// TwinCAT 3 PLC project AdsStaticNetId
// ProgramVersion: 3.1.4023.0
// libraries:
//   Tc2_DataExchange, * (Beckhoff Automation GmbH)
//   Tc2_Standard, * (Beckhoff Automation GmbH)
//   Tc2_System, * (Beckhoff Automation GmbH)
//   Tc2_Utilities, * (Beckhoff Automation GmbH)
//   Tc3_BA_Common, * (Beckhoff Automation GmbH)
//   Tc3_Module, * (Beckhoff Automation GmbH)
// project tree:
//   DUTs/ AdsData.TcDUT (not stored), AdsMessageQueue.TcPOU, AdsMessage.TcDUT (not stored), AdsSocket.TcPOU, AreaNum.TcDUT (not stored), EventsEnum.TcTLEO (not stored)
//   GVLs/ LocalSocket.TcGVL (not stored)
//   / PlcTask.TcTTO (not stored)
//   POUs/ AdsTcp_WinStd.TcPOU, BufferIsEmpty.TcPOU, MAIN.TcPOU
// real-time tasks:
//   TASK PlcTask: cycle T#10ms, priority 21, ADS port 350

// ---- DUTs/AdsMessageQueue.TcPOU
{attribute 'call_after_init'}
FUNCTION_BLOCK AdsMessageQueue
VAR
	elements : FB_BA_DynamicArray := (uiEntrySize := SIZEOF(POINTER TO AdsMessage), uiMinExpCount := 4); 
	length : INT := 0;
	
	entrySize : UDINT;
END_VAR
(*
this container stores dynamically generated AdsData Structs
AdsData to be added are passed by reference, then this function block allocates a structure to be stored
AdsData are get() by reference and poll() by value
*)

METHOD clear : BOOL
VAR
	i : INT;
	temp : REFERENCE TO AdsMessage;
	tempAdr : POINTER TO AdsMessage;
END_VAR
FOR i:=0 TO length-1 BY 1 DO
	temp := get(index := i, getSize => );
	tempAdr := ADR(temp);
	__DELETE(tempAdr);
END_FOR

elements.Reset();
length := 0;
END_METHOD

METHOD contains : BOOL //check contents, not pointer value
VAR_INPUT
	value : REFERENCE TO AdsMessage;
END_VAR
VAR_OUTPUT
	atIndex : INT;
END_VAR
VAR
	temp : REFERENCE TO AdsMessage;
	i : INT;
END_VAR
IF length = 0 THEN
	contains := FALSE;
	RETURN;
END_IF

FOR i:=0 TO length-1 BY 1 DO
	temp := get(index := i, getSize => );
	
	IF 
		SIZEOF(value) = entrySize AND //same size
		MEMCMP(ADR(temp), ADR(value), SIZEOF(entrySize)) = 0 //same data
	THEN
		contains := TRUE;
		atIndex := i;
		RETURN;
	END_IF
	
END_FOR
contains := FALSE;
END_METHOD

METHOD get : REFERENCE TO AdsMessage
VAR_INPUT
	index : INT;
END_VAR
VAR_OUTPUT
	getSize : UDINT;
END_VAR
IF length = 0 OR index < 0 OR index >= length THEN
	getSize := 0;
ELSE
	elements.GetEntry(diIndex := index, pResultEntry := ADR(get));
	getSize := SIZEOF(get);
END_IF
END_METHOD

METHOD isEmpty : BOOL
VAR_INPUT
END_VAR
isEmpty := length = 0;
END_METHOD

METHOD poll : AdsMessage
VAR_OUTPUT
	getSize : UDINT;
END_VAR
IF length > 0 THEN
	poll := get(index := 0, getSize => getSize);
	elements.RemoveEntry(diIndex := 0);
	
	length := length - 1;
END_IF
END_METHOD

METHOD push : BOOL
VAR_INPUT
	value : REFERENCE TO AdsMessage;
END_VAR
VAR
	temp : POINTER TO AdsMessage;
END_VAR
temp := __NEW(AdsMessage);
temp^ := value;

elements.AddEntryPtr(pEntry := temp);

length := length + 1;
END_METHOD

METHOD set : BOOL
VAR_INPUT
	i : INT;
	value : REFERENCE TO AdsMessage;
END_VAR
VAR
	temp : REFERENCE TO AdsMessage;
END_VAR
IF length = 0 THEN
	RETURN;
END_IF

IF i >= 0 AND i < length THEN
	temp REF= get(i);
	temp := value;
	
	set := TRUE;
END_IF
END_METHOD

{attribute 'call_after_init'}
METHOD setup : BOOL
VAR_INPUT
END_VAR
entrySize := SIZEOF(AdsMessage);
END_METHOD

METHOD size : INT
size := length;
END_METHOD

END_FUNCTION_BLOCK

// ---- DUTs/AdsSocket.TcPOU
FUNCTION_BLOCK AdsSocket
VAR_INPUT
END_VAR
VAR_OUTPUT
	//descriptive string for the name of the running program, may or may not be used
	PrgName : STRING;
	
	(*
	AmsNetId should be in the following format for ALL Beckhoff PLCs in the network:
		<area number> . <subarea number (0 for master PLC)> .131.216.1.1
		panel PCs to be assigned 113.174 instead of 131.216
			2.0.131.216.1.1 - Area 2, master controller
			4.3.113.174.1.1 - Area 4, manual station 3 panel PC
	*)
	AmsNetId : T_AmsNetId;
	
	//for now, use ADS port 851 for communication
	AmsPort : T_AmsPort;
END_VAR
VAR_OUTPUT
	receivingData : AdsData;
	sendingData : AdsData;
	
	readBusy : BOOL;
	readError : BOOL;
	readErrorId : UDINT;
	
	writeBusy : BOOL;
	writeError : BOOL;
	writeErrorId : UDINT;
END_VAR
VAR	
	adsWriteSymbol : FB_WriteAdsSymByName;
	adsReadSymbol : FB_ReadAdsSymByName;
END_VAR
VAR
	targetSocket : STRING;
	clearing : BOOL;
END_VAR
(*
TCP-style ADS connection that only writes to a buffer in the recipient's AdsTcpUnit module
*)

//write into the recipient's allocated socket for this system
(*
IF FIND(AmsNetId, '113.174') > 0 THEN //panel PC
	targetSocket := CONCAT('AdsTcp_WinCE.', LocalSocket.PrgName);
ELSE//CX5130+ IPC
	targetSocket := CONCAT('AdsTcp_WinStd.', LocalSocket.PrgName);
END_IF
*)
targetSocket := CONCAT('AdsTcp_WinCE.', LocalSocket.PrgName);
//only toggles if data has contents, otherwise remains false
adsWriteSymbol.bWrite := NOT BufferIsEmpty(sendingData.binaryData) AND NOT adsWriteSymbol.bWrite;
(*
IF NOT BufferIsEmpty(sendingData.binaryData) THEN
	adsWriteSymbol.bWrite := NOT adsWriteSymbol.bWrite;
ELSE
	adsWriteSymbol.bWrite := FALSE;
END_IF 
*)
blocks();

IF NOT adsWriteSymbol.bBusy THEN
	MEMSET(ADR(sendingData), 0, SIZEOF(sendingData));
END_IF

METHOD PRIVATE blocks : BOOL
VAR_INPUT
END_VAR
adsReadSymbol(
	bRead:= , 
	sNetId:= AmsNetId, 
	nPort:= AmsPort, 
	sVarName:= , 
	nDestAddr:= , 
	nLen:= , 
	tTimeout:= , 
	eComMode:= , 
	bClearOnError:= , 
	bBusy=> readBusy, 
	bError=> readError, 
	nErrorId=> readErrorId);
	
adsWriteSymbol(
	bWrite:= , 
	sNetId:= AmsNetId, 
	nPort:= AmsPort, 
	sVarName:= CONCAT(targetSocket, '.receivingData'), 
	nSrcAddr:= ADR(sendingData), 
	nLen:= SIZEOF(sendingData), 
	tTimeout:= , 
	eComMode:= eAdsComModeSecureCom, 
	bBusy=> writeBusy, 
	bError=> writeError, 
	nErrorId=> writeErrorId);
END_METHOD

METHOD send : BOOL
VAR_INPUT
	data : REFERENCE TO AdsData;
END_VAR
sendingData := data;
END_METHOD

END_FUNCTION_BLOCK

// ---- POUs/BufferIsEmpty.TcPOU
FUNCTION BufferIsEmpty : BOOL
VAR_IN_OUT
	bufferArr : ARRAY[*] OF BYTE;
END_VAR
VAR
	i : DINT;
END_VAR

FOR i:=LOWER_BOUND(bufferArr, 1) TO UPPER_BOUND(bufferArr, 1) BY 1 DO
	IF bufferArr[i] <> 0 THEN
		BufferIsEmpty := FALSE;
		RETURN;
	END_IF
END_FOR
BufferIsEmpty := TRUE;

END_FUNCTION

// ---- POUs/AdsTcp_WinStd.TcPOU
PROGRAM AdsTcp_WinStd
VAR_OUTPUT
	bBusy : BOOL;
	err : BOOL;
	errid : UDINT;
END_VAR
VAR_OUTPUT
	areaSockets : ARRAY[1..6] OF POINTER TO AdsSocket; //only used for finding a socket by name, POINTER because array of REFERENCE does not exist
	
	//unlikely that each area will need communication with all other areas
	//only area 3 needs access to all areas, other areas only need access to area 3
	AREA_1 : AdsSocket := (PrgName := 'AREA_1', AmsNetId := '1.0.131.216.1.1', AmsPort := 851);
	AREA_2 : AdsSocket := (PrgName := 'AREA_2', AmsNetId := '2.0.131.216.1.1', AmsPort := 851);
	AREA_3 : AdsSocket := (PrgName := 'AREA_3', AmsNetId := '3.0.131.216.1.1', AmsPort := 851);
	AREA_4 : AdsSocket := (PrgName := 'AREA_4', AmsNetId := '4.0.131.216.1.1', AmsPort := 851);
	AREA_5 : AdsSocket := (PrgName := 'AREA_5', AmsNetId := '5.0.131.216.1.1', AmsPort := 851);
	AREA_6 : AdsSocket := (PrgName := 'AREA_6', AmsNetId := '6.0.131.216.1.1', AmsPort := 851);
END_VAR
VAR	
	tempSocket : REFERENCE TO AdsSocket;
	(*
	transmissons are queued into AdsTcpUnit, where all the preset sockets are
	to send a transmission, place the data and a recipient name into an AdsMessage type
	when a transmission is polled from the queue:
		if the recipient does not exist, the message contents are discarded
		if the recipient exists and is not busy writing, then the message contents are given to the socket to be written
		if the recipient is busy, then the messsage is pushed back into the queue
	*)
	transmissionQueue : AdsMessageQueue;
	nextTransmission : AdsMessage;
	
	i : INT(1..numSockets);
END_VAR
VAR CONSTANT
	numSockets : INT := 6-1;
END_VAR
(*
similar functionality to standard TCP communication - only writes to a single receiving buffer on the target system
	no read/write functionality to any other symbol on target
messages are entered into a queue which is polled cyclically and passed to the appropriate socket
*)

areaSockets[1] := ADR(AREA_1);
areaSockets[2] := ADR(AREA_2);
areaSockets[3] := ADR(AREA_3);
areaSockets[4] := ADR(AREA_4);
areaSockets[5] := ADR(AREA_5);
areaSockets[6] := ADR(AREA_6);

blocks();

nextTransmission := transmissionQueue.poll(getSize => );

tempSocket REF= findSocket(recipient := nextTransmission.recipient);

IF __ISVALIDREF(tempSocket) THEN
	
	IF NOT tempSocket.writeBusy THEN
		tempSocket.send(data := nextTransmission.contents);
	ELSE //if socket is busy, then message is returned to the end of the line
		transmissionQueue.push(value := nextTransmission);
	END_IF
	
END_IF
//if recipient does not exist, message is discarded

METHOD PRIVATE blocks : BOOL
VAR_INPUT
END_VAR
AREA_1(
	PrgName=> , 
	AmsNetId=> , 
	AmsPort=> , 
	receivingData=> , 
	sendingData=> , 
	readBusy=> , 
	readError=> , 
	readErrorId=> , 
	writeBusy=> , 
	writeError=> , 
	writeErrorId=> );

AREA_2(
	PrgName=> , 
	AmsNetId=> , 
	AmsPort=> , 
	receivingData=> , 
	sendingData=> , 
	readBusy=> , 
	readError=> , 
	readErrorId=> , 
	writeBusy=> , 
	writeError=> , 
	writeErrorId=> );
	
AREA_3(
	PrgName=> , 
	AmsNetId=> , 
	AmsPort=> , 
	receivingData=> , 
	sendingData=> , 
	readBusy=> , 
	readError=> , 
	readErrorId=> , 
	writeBusy=> , 
	writeError=> , 
	writeErrorId=> );
	
AREA_4(
	PrgName=> , 
	AmsNetId=> , 
	AmsPort=> , 
	receivingData=> , 
	sendingData=> , 
	readBusy=> , 
	readError=> , 
	readErrorId=> , 
	writeBusy=> , 
	writeError=> , 
	writeErrorId=> );
	
AREA_5(
	PrgName=> , 
	AmsNetId=> , 
	AmsPort=> , 
	receivingData=> , 
	sendingData=> , 
	readBusy=> , 
	readError=> , 
	readErrorId=> , 
	writeBusy=> , 
	writeError=> , 
	writeErrorId=> );
	
AREA_6(
	PrgName=> , 
	AmsNetId=> , 
	AmsPort=> , 
	receivingData=> , 
	sendingData=> , 
	readBusy=> , 
	readError=> , 
	readErrorId=> , 
	writeBusy=> , 
	writeError=> , 
	writeErrorId=> );
END_METHOD

METHOD PRIVATE findSocket : REFERENCE TO AdsSocket
VAR_INPUT
	recipient : STRING;
END_VAR
FOR i:=1 TO numSockets BY 1 DO
	IF areaSockets[i]^.PrgName = recipient THEN
		findSocket REF= areaSockets[i]^;
		RETURN;
	END_IF
END_FOR
END_METHOD

METHOD generateMessage : BOOL
VAR_INPUT
	recipient : STRING;
	description : EventsEnum;
	timestamp : TIMESTRUCT;
END_VAR
VAR_IN_OUT
	binaryData : ARRAY[*] OF BYTE;
END_VAR
VAR
	newTransmission : AdsMessage;
END_VAR
newTransmission.recipient := recipient;

newTransmission.contents.description := description;
newTransmission.contents.timestamp := timestamp;
MEMCPY(
	ADR(newTransmission.contents.binaryData),
	binaryData,
	MIN( TO_UDINT(UPPER_BOUND(binaryData, 1) - LOWER_BOUND(binaryData, 1) + 1), SIZEOF(newTransmission.contents.binaryData) ));
END_METHOD

METHOD pollData : BOOL
VAR_INPUT
	//remotePrgName : STRING;
	buffer : PVOID;
	bufferSize : UDINT;
	
	data : PVOID;
	dataSize : UDINT;
END_VAR
MEMCPY(buffer, data, MIN(dataSize, bufferSize));
MEMSET(data, 0, dataSize);
END_METHOD

METHOD queueMessage : BOOL
VAR_INPUT
	recipient : STRING;
	data : REFERENCE TO AdsData;
END_VAR
VAR
	newMessage : AdsMessage;
END_VAR
IF recipient <> '' THEN
	newMessage.recipient := recipient;
	newMessage.contents := data;
	
	transmissionQueue.push(newMessage);
	
	queueMessage := TRUE;
END_IF
END_METHOD

METHOD retrieveData : BOOL
VAR_INPUT
	name : STRING;
END_VAR
VAR_IN_OUT
	genericBuffer : ARRAY[*] OF BYTE;
END_VAR
VAR
	bufferSize : DINT;
	
	//reqHandle : REFERENCE TO AdsHandle;
END_VAR
(*
bufferSize := UPPER_BOUND(genericBuffer, 1) - LOWER_BOUND(genericBuffer, 1) + 1;

reqHandle REF= findHandle('CLIENT_1');

IF __ISVALIDREF(reqHandle) THEN
	genericBuffer := ADR(reqHandle.genericBuffer);
	stDemo := reqHandle.receiverStDemo;
END_IF
*)
END_METHOD

END_PROGRAM

// ---- POUs/MAIN.TcPOU
PROGRAM MAIN
VAR_OUTPUT
	currentTime : TIMESTRUCT;
END_VAR
VAR
	sMessage : STRING := 'from SERVER to CLIENT';
	newRecipient : STRING;
	newData : AdsData;
	retrievedData : AdsData;
	
	sendOnce : BOOL;
	sendFastNum : BOOL;
	
	i : INT := 0;
	
	fbLocalSystemTime : FB_LocalSystemTime;
END_VAR

IF NOT setup() THEN
	RETURN;
END_IF

AdsTcp_WinStd(
	bBusy=> , 
	err=> , 
	errid=> , 
	areaSockets=> );
	
IF sendOnce OR sendFastNum THEN
	MEMSET(ADR(newData), 0, SIZEOF(newData));
	
	sMessage := TO_STRING(i);
	
	newRecipient := TO_STRING(AreaNum.AREA_2);
	newData.description := EventsEnum.TEST_COMMS;
	newData.timestamp := currentTime;
	MEMCPY(ADR(newData.binaryData), ADR(sMessage), LEN(sMessage));
	
	AdsTcp_WinStd.queueMessage(recipient := newRecipient, data := newData);
	
	i := i + 1;
	sendOnce := FALSE;
END_IF

retrievedData := AdsTcp_WinStd.AREA_2.receivingData;

METHOD setup : BOOL
VAR
END_VAR
fbLocalSystemTime(
	sNetID:= , 
	bEnable:= TRUE, 
	dwCycle:= , 
	dwOpt:= , 
	tTimeout:= , 
	bValid=> , 
	systemTime=> currentTime, 
	tzID=> );

setup := TRUE;
END_METHOD

END_PROGRAM
